RoboDK station: Conveying-with-UR10 (1).rdk

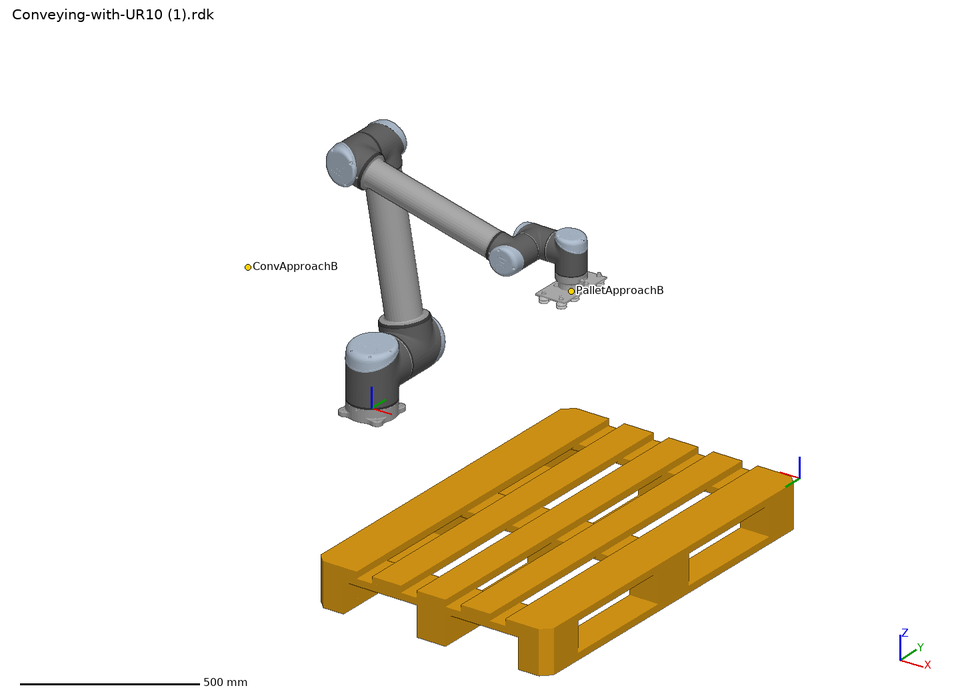
[picture v0: the station drawn from its stored meshes, robots at their saved joint values, targets as dots, program paths as lines]
Station Conveying with UR10 (saved by RoboDK 6.0.5). Poses are relative to the parent item; angles as X-Y-Z fixed-axis rotations.
Station parameters (name, value as stored): SizeBox, 150, 200, 150, SizePallet, 3,2,3, ConvSpeed, 25.0, SENSOR, 0
  - notes Description: <!DOCTYPE HTML PUBLIC "-//W3C//DTD HTML 4.0//EN" "http://www.w3.org/TR/REC-html40/strict.dtd">
<html><head><meta name="qrichtext" content="1" /><style type="text/css">
p, li { white-space: pre-wrap; }
</style></head><body style=" font-family:'MS Shell Dlg 2'; font-size:8.25pt; font-weight:400; font-style:normal;">
<p style=" margin-top:0px; margin-bottom:0px; margin-left:0px; margin-right:0px; -qt-block-indent:0; text-indent:0px;">This example demonstrates a dual-robot pick-and-place application using two collaborative 6-axis UR10 robots equipped with suction cup grippers. The first robot picks cubes from a pallet and places them onto a continuously moving conveyor. The second robot picks the cubes from the conveyor and places them onto another pallet. A Python script developed with the RoboDK API simulates the detection of the cubes on the moving conveyor before the second robot performs the pick operation.</p></body></html>
  - frame UR10 Base B at (1478.64, 1242.75, 0) mm
    - robot UR10 B (model UR10): 6 axes, payload 10 kg, reach 1300 mm, repeatability 0.1 mm, weight 28.9 kg
        modified DH rows (alpha deg, a mm, theta deg, d mm): 0, 0, 0, 118; 90, 0, 180, 0; 0, 612.7, 0, 0; 0, 571.6, 0, 163.9; -90, 0, 0, 115.7; 90, 0, 180, 92.2
        joint limits [-360, -360, -360, -360, -360, -360] to [360, 360, 360, 360, 360, 360]; home [0, -90, 90, -90, -90, 0]; saved at [-180.64, -99.905, 114.086, -104.182, -90, 0]
      - tool GripperB, TCP at (0, 0, 30) mm, rotated rx 0 ry 0 rz 90 deg, size 209.9 x 42 x 100 mm, geometry from test.iges
    - target ConvApproachB (joint target) at (-305.88, -163.9, 417.02) mm, rotated rx -180 ry 0 rz 0 deg; joints [0, -128.114, 134.225, -96.111, -90, 0] of UR10 B
    - target PalletApproachB (joint target) at (566.28, 157.58, 459.33) mm, rotated rx -180 ry 0 rz 179.36 deg; joints [-180.64, -99.905, 114.086, -104.182, -90, 0] of UR10 B
    - frame PalletB at (1034.81, 598.47, -166.38) mm, rotated rx 0 ry 0 rz 179.17 deg
      - object Europallet at (0, 0, 0) mm, size 800 x 144 x 1200 mm, geometry from UUID&
  - program MoveConveyor (1 instructions, listed below)
  - program MainSimulation (5 instructions, listed below)
  - Python program PalletizePreview (listed below)
  - Python program PrepareSimulation (listed below)
  - Python program RobotA_GetParts (listed below)
  - Python program RobotB_StoreParts (listed below)
  - Python program SensorActivate (listed below)
  - Python program SetSimulationParams (listed below)

--- program MoveConveyor ---
  MoveJ (ConveyorMove) [its target is no longer in the station]

--- program MainSimulation ---
  Call PrepareSimulation
  Run MoveConveyor
  Run RobotA_GetParts
  Run SensorActivate
  Call RobotB_StoreParts

--- Python program PalletizePreview ---
# PalletizePreview — roda DENTRO do RoboDK e paletiza com ciclo pick -> place real.
#
# O pick e feito na ESTEIRA (Get Conveyor / ConvApproach), do lado oposto ao pallet, como no
# RobotB_StoreParts.py: a caixa surge sobre a esteira, o robo PEGA (a caixa segue a garra),
# leva ao pallet e SOLTA, camada por camada. Padroes (grid/brick/pinhole/split_block) sao os
# mesmos de palletizer/planner/patterns.py.
#
# COMO RODAR: arraste este arquivo para a janela do RoboDK (ou Tools > Run Script) e Play.

from robodk import robolink, robomath

# ----------------------------- AJUSTE AQUI -----------------------------
PATTERN = "brick"        # "grid" | "brick" | "pinhole" | "split_block"
LAYERS = 4               # no de camadas (minimo 2)
ROBOT_LETTER = "B"       # "A" ou "B" (qual UR10 da estacao)
MOVE_ROBOT = True        # False = so preenche o pallet, sem pick nem robo
APPROACH = 100.0         # folga de aproximacao vertical (mm)

# Nomes da esteira na estacao (fonte do pick). Ajuste se forem diferentes.
CONV_FRAME = "ConveyorReference"
CONV_TARGET = "Get Conveyor"        # ponto de coleta sobre a esteira
CONV_APPROACH = "ConvApproach"      # + letra do robo (ex.: ConvApproachB)

# Fallback (usado SO se a esteira nao for encontrada): pick ao lado do pallet.
PICK_DX = None           # None = centro do pallet em X
PICK_DY = -150.0
# -----------------------------------------------------------------------

RDK = robolink.Robolink()
RDK.setRunMode(robolink.RUNMODE_SIMULATE)


# =========== padroes de amarracao (espelho de planner/patterns.py) ===========
def _base_grid(nx, ny, bx, by):
    return [((i + 0.5) * bx, (j + 0.5) * by, 0.0)
            for j in range(ny) for i in range(nx)]


def layer_positions(pattern, nx, ny, bx, by, layer):
    pos = _base_grid(nx, ny, bx, by)
    if pattern == "brick":
        if layer % 2 == 1:
            pos = [(x + bx / 2.0, y, r) for (x, y, r) in pos]
    elif pattern == "pinhole":
        center = round((ny - 1) / 2.0) * nx + round((nx - 1) / 2.0)
        pos = [p for k, p in enumerate(pos) if k != center]
        if layer % 2 == 1:
            pos = [(x, y, (r + 90.0) % 180.0) for (x, y, r) in pos]
    elif pattern == "split_block":
        mid = nx / 2.0
        pos = [(x, y, 90.0 if ((k % nx < mid) == (layer % 2 == 1)) else 0.0)
               for k, (x, y, r) in enumerate(pos)]
    return pos


# =========== geometria a partir dos params da estacao ===========
def _parse_triplet(value, default):
    try:
        parts = [float(v.replace(" ", "")) for v in str(value).split(",")]
        if len(parts) >= 3:
            return parts[:3]
    except Exception:
        pass
    return default


BX, BY, BZ = _parse_triplet(RDK.getParam("SizeBox"), [100.0, 100.0, 100.0])
size_pallet = _parse_triplet(RDK.getParam("SizePallet"), [3.0, 3.0, float(LAYERS)])
NX, NY = int(size_pallet[0]), int(size_pallet[1])


# =========== itens da estacao ===========
suffix = ROBOT_LETTER.upper()
robot = RDK.Item("UR10 " + suffix, robolink.ITEM_TYPE_ROBOT)
tool = RDK.Item("Gripper" + suffix, robolink.ITEM_TYPE_TOOL)
frame_pallet = RDK.Item("Pallet" + suffix, robolink.ITEM_TYPE_FRAME)
target_safe = RDK.Item("PalletApproach" + suffix, robolink.ITEM_TYPE_TARGET)
partref = RDK.Item("box100mm")

for label, item in [("UR10 " + suffix, robot), ("Pallet" + suffix, frame_pallet),
                    ("box100mm", partref)]:
    if not item.Valid():
        raise Exception("Item '%s' nao encontrado na estacao. Ajuste os nomes no topo." % label)

# esteira (fonte do pick)
frame_conv = RDK.Item(CONV_FRAME, robolink.ITEM_TYPE_FRAME)
target_conv = RDK.Item(CONV_TARGET, robolink.ITEM_TYPE_TARGET)
conv_safe = RDK.Item(CONV_APPROACH + suffix, robolink.ITEM_TYPE_TARGET)
use_conveyor = frame_conv.Valid() and target_conv.Valid()

has_pallet_safe = target_safe.Valid()

# --- define onde e como fazer o pick ---
if use_conveyor:
    pick_frame = frame_conv
    pick_safe = conv_safe if conv_safe.Valid() else None
    pick_tool = target_conv.Pose() * robomath.transl(0, 0, -BZ / 2.0)  # pose de coleta na esteira
    box_local = robomath.transl(*pick_tool.Pos())                      # caixa upright sobre a esteira
    print("Pick: ESTEIRA ('%s')." % CONV_TARGET)
else:
    pick_frame = frame_pallet
    pick_safe = target_safe if has_pallet_safe else None
    px = (NX * BX / 2.0) if PICK_DX is None else PICK_DX
    pick_tool = robomath.transl(px, PICK_DY, BZ / 2.0) * robomath.rotx(robomath.pi)
    box_local = robomath.transl(px, PICK_DY, BZ / 2.0)
    print("Pick: esteira nao encontrada; usando ponto ao lado do pallet (%.0f, %.0f)."
          % (px, PICK_DY))

pick_app = pick_tool * robomath.transl(0, 0, -(APPROACH + BZ))


# =========== limpa caixas anteriores ===========
RDK.Render(False)
for obj in RDK.ItemList(robolink.ITEM_TYPE_OBJECT, False):
    if obj.Name().startswith("Caixa "):
        obj.Delete()
partref.Copy()

if MOVE_ROBOT and tool.Valid():
    robot.setPoseTool(tool)


# =========== helpers ===========
def new_box(index, layer):
    part = frame_pallet.Paste()
    part.Scale([BX / 100.0, BY / 100.0, BZ / 100.0])
    part.setName("Caixa %d" % index)
    part.Recolor([0.2, 0.5, 0.2 + 0.6 * (layer % 2), 1])
    part.setVisible(True, False)
    return part


def rotz(deg):
    return robomath.rotz(robomath.pi * deg / 180.0)


def snap(part, x, y, z, rot_z):
    part.setParentStatic(frame_pallet)
    part.setPose(robomath.transl(x, y, z) * rotz(rot_z))


# =========== execucao ===========
count = 0
reach_fail = 0
first_error_shown = False
for layer in range(LAYERS):
    z_center = (layer + 0.5) * BZ
    for (x, y, rot_z) in layer_positions(PATTERN, NX, NY, BX, BY, layer):
        count += 1
        part = new_box(count, layer)

        if not MOVE_ROBOT:
            snap(part, x, y, z_center, rot_z)
            continue

        # a caixa surge no ponto de coleta (esteira)
        part.setParent(pick_frame)
        part.setPose(box_local)
        RDK.Render(True)

        place = robomath.transl(x, y, z_center) * robomath.rotx(robomath.pi) * rotz(rot_z)
        place_app = place * robomath.transl(0, 0, -(APPROACH + BZ))

        try:
            # PEGA na esteira
            robot.setPoseFrame(pick_frame)
            if pick_safe is not None:
                robot.MoveJ(pick_safe)
            robot.MoveJ(pick_app)
            robot.MoveL(pick_tool)
            part.setParentStatic(tool)      # anexa a caixa a garra
            robot.MoveL(pick_app)
            # SOLTA no pallet
            robot.setPoseFrame(frame_pallet)
            if has_pallet_safe:
                robot.MoveJ(target_safe)
            robot.MoveJ(place_app)
            robot.MoveL(place)
            snap(part, x, y, z_center, rot_z)  # encaixa exato
            robot.MoveL(place_app)
        except Exception as exc:
            reach_fail += 1
            snap(part, x, y, z_center, rot_z)
            if not first_error_shown:
                print("ERRO de movimento na caixa %d: %s" % (count, exc))
                print("  -> verifique alcance do pick/place ou os nomes da esteira no topo.")
                first_error_shown = True

if MOVE_ROBOT and has_pallet_safe:
    try:
        robot.setPoseFrame(frame_pallet)
        robot.MoveJ(target_safe)
    except Exception:
        pass

RDK.Render(True)
print("Padrao '%s': %d caixas, %d camada(s), %d falha(s) de alcance."
      % (PATTERN, count, LAYERS, reach_fail))

--- Python program PrepareSimulation ---
# Type help("robodk.robolink") or help("robodk.robomath") for more information
# Press F5 to run the script
# Documentation: https://robodk.com/doc/en/RoboDK-API.html
# Reference:     https://robodk.com/doc/en/PythonAPI/robodk.html
# Note: It is not required to keep a copy of this file, your Python script is saved with your RDK project

# You can also use the new version of the API:
from robodk import robolink    # RoboDK API
from robodk import robomath    # Robot toolbox
RDK = robolink.Robolink()

# Forward and backwards compatible use of the RoboDK API:
# Remove these 2 lines to follow python programming guidelines
from robodk import *      # RoboDK API
from robolink import *    # Robot toolbox
# Link to RoboDK
# RDK = Robolink()
# Type help("robolink") or help("robodk") for more information
# Press F5 to run the script
# Note: you do not need to keep a copy of this file, your python script is saved with the station

# Use RoboDK API as RL

frame_pallet        = RDK.Item('PalletA', robolink.ITEM_TYPE_FRAME)

# get variable parameters
SIZE_BOX = RDK.getParam('SizeBox')
SIZE_PALLET = RDK.getParam('SizePallet')
SIZE_BOX_XYZ = [float(x.replace(' ','')) for x in SIZE_BOX.split(',')]
SIZE_PALLET_XYZ = [float(x.replace(' ','')) for x in SIZE_PALLET.split(',')]
SIZE_BOX_Z = SIZE_BOX_XYZ[2] # the height of the boxes is important to take into account when approaching the positions

def box_calc(size_xyz, pallet_xyz):
    """Calculates a list of points to store parts in a pallet"""
    [size_x, size_y, size_z] = size_xyz
    [pallet_x, pallet_y, pallet_z] = pallet_xyz
    xyz_list = []
    for h in range(int(pallet_z)):
        for j in range(int(pallet_y)):
            for i in range(int(pallet_x)):
                xyz_list = xyz_list + [[(i+0.5)*size_x, (j+0.5)*size_y, (h+0.5)*size_z]]
    return xyz_list

def parts_setup(frame, positions, size_xyz):
    """Place a list of parts in a reference frame. The part/reference object must have been previously copied to the clipboard."""
    [size_x, size_y, size_z] = size_xyz
    nparts = len(positions)
    cstep = 1.0/(nparts - 1)
    for i in range(nparts):
        newpart = frame.Paste()
        newpart.Scale([size_x/100, size_y/100, size_z/100]) #scale with respect to the reference object (100mm cube)
        newpart.setName('Part ' + str(i+1)) #set item name
        newpart.setPose(robomath.transl(positions[i])) #set item position with respect to parent
        newpart.setVisible(True, False) #make item visible but hide the reference frame
        newpart.Recolor([1-cstep*i, cstep*i, 0.2, 1]) #set RGBA color

def cleanup(objects, startswith="Part "):
    """Deletes all objects where the name starts with "startswith", from the provided list of objects."""
    for item in objects:
        if item.Name().startswith(startswith):
            item.Delete()

# turn off rendering (much faster when setting up the station)
RDK.Render(False)

# cleanup previous simulation (generated parts and tools)
all_objects = RDK.ItemList(robolink.ITEM_TYPE_OBJECT, False)
cleanup(all_objects, 'Part ')
all_tools = RDK.ItemList(robolink.ITEM_TYPE_TOOL, False)
cleanup(all_tools, 'TCP ')

# copy the reference part
partref = RDK.Item('box100mm')
partref.Copy()

#RL.Set_Simulation_Speed(500);
#RL.Set_Simulation_Mode(1)

# calculate an array of positions to get/store the parts
parts_positions = box_calc(SIZE_BOX_XYZ, SIZE_PALLET_XYZ)

# setup/initialise the parts on the palled
parts_setup(frame_pallet, parts_positions, SIZE_BOX_XYZ)

RDK.Render(True)

--- Python program RobotA_GetParts ---
# Type help("robodk.robolink") or help("robodk.robomath") for more information
# Press F5 to run the script
# Documentation: https://robodk.com/doc/en/RoboDK-API.html
# Reference:     https://robodk.com/doc/en/PythonAPI/robodk.html
# Note: It is not required to keep a copy of this file, your Python script is saved with your RDK project

# You can also use the new version of the API:
from robodk import robolink    # RoboDK API
from robodk import robomath    # Robot toolbox
RDK = robolink.Robolink()

# Forward and backwards compatible use of the RoboDK API:
# Remove these 2 lines to follow python programming guidelines
from robodk import *      # RoboDK API
from robolink import *    # Robot toolbox
# Link to RoboDK
# RDK = Robolink()
# Type help("robolink") or help("robodk") for more information
# Press F5 to run the script
# Note: you do not need to keep a copy of this file, your python script is saved with the station

# Use RoboDK API as RL

# define default approach distance
APPROACH = 100

# gather robot, tool and reference frames from the station
robot               = RDK.Item('UR10 A', robolink.ITEM_TYPE_ROBOT)
tool                = RDK.Item('GripperA', robolink.ITEM_TYPE_TOOL)
frame_pallet        = RDK.Item('PalletA', robolink.ITEM_TYPE_FRAME)
frame_conv          = RDK.Item('ConveyorReference', robolink.ITEM_TYPE_FRAME)
frame_conv_moving   = RDK.Item('MovingRef', robolink.ITEM_TYPE_FRAME)

# gather targets
target_pallet_safe = RDK.Item('PalletApproachA', robolink.ITEM_TYPE_TARGET)
target_conv_safe = RDK.Item('ConvApproachA', robolink.ITEM_TYPE_TARGET)
target_conv = RDK.Item('Put Conveyor', robolink.ITEM_TYPE_TARGET)

# get variable parameters
SIZE_BOX = RDK.getParam('SizeBox')
SIZE_PALLET = RDK.getParam('SizePallet')
SIZE_BOX_XYZ = [float(x.replace(' ','')) for x in SIZE_BOX.split(',')]
SIZE_PALLET_XYZ = [float(x.replace(' ','')) for x in SIZE_PALLET.split(',')]
SIZE_BOX_Z = SIZE_BOX_XYZ[2] # the height of the boxes is important to take into account when approaching the positions

def box_calc(size_xyz, pallet_xyz):
    """Calculates a list of points to store parts in a pallet"""
    [size_x, size_y, size_z] = size_xyz
    [pallet_x, pallet_y, pallet_z] = pallet_xyz
    xyz_list = []
    for h in range(int(pallet_z)):
        for j in range(int(pallet_y)):
            for i in range(int(pallet_x)):
                xyz_list = xyz_list + [[(i+0.5)*size_x, (j+0.5)*size_y, (h+0.5)*size_z]]
    return xyz_list

def TCP_On(toolitem):
    """Attaches the closest object to the toolitem Htool pose,
    It will also output appropriate function calls on the generated robot program (call to TCP_On)"""
    toolitem.AttachClosest()
    toolitem.RDK().RunMessage('Set air valve on')
    toolitem.RDK().RunProgram('TCP_On()');

def TCP_Off(toolitem, itemleave=0):
    """Detaches the closest object attached to the toolitem Htool pose,
    It will also output appropriate function calls on the generated robot program (call to TCP_Off)"""
    toolitem.DetachAll(itemleave)
    toolitem.RDK().RunMessage('Set air valve off')
    toolitem.RDK().RunProgram('TCP_Off()');

#RL.Set_Simulation_Speed(500);
#RL.Set_Simulation_Mode(1)

# calculate an array of positions to get/store the parts
parts_positions = box_calc(SIZE_BOX_XYZ, SIZE_PALLET_XYZ)

# Calculate a new TCP that takes into account the size of the part (targets are set to the center of the box)
tool_xyzrpw = tool.PoseTool()*robomath.transl(0,0,SIZE_BOX_Z/2)
tool_tcp = robot.AddTool(tool_xyzrpw, 'TCP A')

# ---------------------------------------------------------------------------------
# -------------------------- PROGRAM START ----------------------------------------

robot.setPoseTool(tool_tcp)
nparts = len(parts_positions)
i = nparts-1
while i >= 0:
    # ----------- take a part from the pallet ------
    # get the xyz position of part i
    robot.setPoseFrame(frame_pallet)
    part_position_i = parts_positions[i]
    target_i = robomath.transl(part_position_i)*robomath.rotx(pi)
    target_i_app = target_i * robomath.transl(0,0,-(APPROACH+SIZE_BOX_Z))
    # approach to the pallet
    robot.MoveJ(target_pallet_safe)
    # get the box i
    robot.MoveJ(target_i_app)
    robot.MoveL(target_i)
    TCP_On(tool) # attach the closest part
    robot.MoveL(target_i_app)
    robot.MoveJ(target_pallet_safe)

    # ----------- place the box i on the convegor ------
    # approach to the conveyor
    robot.setPoseFrame(frame_conv)
    target_conv_pose = target_conv.Pose()*robomath.transl(0,0,-SIZE_BOX_Z/2)
    target_conv_app = target_conv_pose*robomath.transl(0,0,-APPROACH)
    robot.MoveJ(target_conv_safe)
    robot.MoveJ(target_conv_app)
    robot.MoveL(target_conv_pose)
    TCP_Off(tool, frame_conv_moving) # detach an place the object in the moving reference frame of the conveyor
    robot.MoveL(target_conv_app)
    robot.MoveJ(target_conv_safe)

    i = i - 1

--- Python program RobotB_StoreParts ---
# Type help("robodk.robolink") or help("robodk.robomath") for more information
# Press F5 to run the script
# Documentation: https://robodk.com/doc/en/RoboDK-API.html
# Reference:     https://robodk.com/doc/en/PythonAPI/robodk.html
# Note: It is not required to keep a copy of this file, your Python script is saved with your RDK project

# You can also use the new version of the API:
from robodk import robolink    # RoboDK API
from robodk import robomath    # Robot toolbox
RDK = robolink.Robolink()

# Forward and backwards compatible use of the RoboDK API:
# Remove these 2 lines to follow python programming guidelines
from robodk import *      # RoboDK API
from robolink import *    # Robot toolbox
# Link to RoboDK
# RDK = Robolink()
# Type help("robolink") or help("robodk") for more information
# Press F5 to run the script
# Note: you do not need to keep a copy of this file, your python script is saved with the station

# Use RoboDK API as RL

# define default approach distance
APPROACH = 100
SENSOR_VARIABLE = 'SENSOR' # station variable

# gather robot, tool and reference frames from the station
robot               = RDK.Item('UR10 B', robolink.ITEM_TYPE_ROBOT)
tool                = RDK.Item('GripperB', robolink.ITEM_TYPE_TOOL)
frame_pallet        = RDK.Item('PalletB', robolink.ITEM_TYPE_FRAME)
frame_conv          = RDK.Item('ConveyorReference', robolink.ITEM_TYPE_FRAME)
frame_conv_moving   = RDK.Item('MovingRef', robolink.ITEM_TYPE_FRAME)

# gather targets
target_pallet_safe = RDK.Item('PalletApproachB', robolink.ITEM_TYPE_TARGET)
target_conv_safe = RDK.Item('ConvApproachB', robolink.ITEM_TYPE_TARGET)
target_conv = RDK.Item('Get Conveyor', robolink.ITEM_TYPE_TARGET)

# get variable parameters
SIZE_BOX = RDK.getParam('SizeBox')
SIZE_PALLET = RDK.getParam('SizePallet')
SIZE_BOX_XYZ = [float(x.replace(' ','')) for x in SIZE_BOX.split(',')]
SIZE_PALLET_XYZ = [float(x.replace(' ','')) for x in SIZE_PALLET.split(',')]
SIZE_BOX_Z = SIZE_BOX_XYZ[2] # the height of the boxes is important to take into account when approaching the positions

def box_calc(size_xyz, pallet_xyz):
    """Calculates a list of points to store parts in a pallet"""
    [size_x, size_y, size_z] = size_xyz
    [pallet_x, pallet_y, pallet_z] = pallet_xyz
    xyz_list = []
    for h in range(int(pallet_z)):
        for j in range(int(pallet_y)):
            for i in range(int(pallet_x)):
                xyz_list = xyz_list + [[(i+0.5)*size_x, (j+0.5)*size_y, (h+0.5)*size_z]]
    return xyz_list

def TCP_On(toolitem):
    """Attaches the closest object to the toolitem Htool pose,
    It will also output appropriate function calls on the generated robot program (call to TCP_On)"""
    toolitem.AttachClosest()
    toolitem.RDK().RunMessage('Set air valve on')
    toolitem.RDK().RunProgram('TCP_On()');

def TCP_Off(toolitem, itemleave=0):
    """Detaches the closest object attached to the toolitem Htool pose,
    It will also output appropriate function calls on the generated robot program (call to TCP_Off)"""
    #toolitem.DetachClosest(itemleave)
    toolitem.DetachAll(itemleave)
    toolitem.RDK().RunMessage('Set air valve off')
    toolitem.RDK().RunProgram('TCP_Off()');

# calculate an array of positions to get/store the parts
parts_positions = box_calc(SIZE_BOX_XYZ, SIZE_PALLET_XYZ)

# Calculate a new TCP that takes into account the size of the part (targets are set to the center of the box)
tool_xyzrpw = tool.PoseTool()*robomath.transl(0,0,SIZE_BOX_Z/2)
tool_tcp = robot.AddTool(tool_xyzrpw, 'TCP B')

# ---------------------------------------------------------------------------------
# -------------------------- PROGRAM START ----------------------------------------

def WaitSensor():
    if RDK.RunMode() == robolink.RUNMODE_SIMULATE:
        # Simulate the sensor by waiting for the SENSOR status to turn to 1 (object present)
        while RDK.getParam(SENSOR_VARIABLE) == 0:
            pause(0.001)
    else:
        RDK.RunProgram('WaitSensor')
    print("Part detected")

robot.setPoseTool(tool_tcp)
nparts = len(parts_positions)
i = 0
while i < nparts:
    # ----------- place the box i on the convegor ------
    # approach to the conveyor
    robot.setPoseFrame(frame_conv)
    target_conv_pose = target_conv.Pose()*robomath.transl(0,0,-SIZE_BOX_Z/2)
    target_conv_app = target_conv_pose*robomath.transl(0,0,-APPROACH)
    robot.MoveJ(target_conv_safe)
    robot.MoveJ(target_conv_app)
    WaitSensor()
    robot.MoveL(target_conv_pose)
    TCP_On(tool) # detach an place the object in the moving reference frame of the conveyor
    robot.MoveL(target_conv_app)
    robot.MoveJ(target_conv_safe)

    # ----------- take a part from the conveyor ------
    # get the xyz position of part i
    robot.setPoseFrame(frame_pallet)
    part_position_i = parts_positions[i]
    target_i = robomath.transl(part_position_i)*robomath.rotx(pi)
    target_i_app = target_i * robomath.transl(0,0,-(APPROACH+SIZE_BOX_Z))
    # approach to the pallet
    robot.MoveJ(target_pallet_safe)
    # get the box i
    robot.MoveJ(target_i_app)
    robot.MoveL(target_i)
    TCP_Off(tool, frame_pallet) # attach the closest part
    robot.MoveL(target_i_app)
    robot.MoveJ(target_pallet_safe)

    i = i + 1

--- Python program SensorActivate ---
# Type help("robodk.robolink") or help("robodk.robomath") for more information
# Press F5 to run the script
# Documentation: https://robodk.com/doc/en/RoboDK-API.html
# Reference:     https://robodk.com/doc/en/PythonAPI/robodk.html
# Note: It is not required to keep a copy of this file, your Python script is saved with your RDK project

# You can also use the new version of the API:
from robodk import robolink    # RoboDK API
from robodk import robomath    # Robot toolbox
RDK = robolink.Robolink()

# Forward and backwards compatible use of the RoboDK API:
# Remove these 2 lines to follow python programming guidelines
from robodk import *      # RoboDK API
from robolink import *    # Robot toolbox
# Link to RoboDK
# RDK = Robolink()
# Type help("robolink") or help("robodk") for more information
# Press F5 to run the script
# Note: you do not need to keep a copy of this file, your python script is saved with the station

# This script allows to simulate a laser sensor
# that detect the presence of a part in a plane,
# such as a part crossing a laser sensor in a
# conveyor belt

# Use a target from the station as a reference plane:
SENSOR_NAME = 'Sensor SICK WL4S'
SENSOR_VARIABLE = 'SENSOR'

# Look for parts with the keyword "Part"
PART_KEYWORD = 'Part '

# Update status every 1 ms
RECHECK_PERIOD = 0.001

# Get the sensor and the detection plane
SENSOR = RDK.Item(SENSOR_NAME, robolink.ITEM_TYPE_OBJECT)

# retrieve all objects
all_objects = RDK.ItemList(robolink.ITEM_TYPE_OBJECT, False)
part_objects = []
for obj in all_objects:
    if obj.Name().count(PART_KEYWORD) > 0:
        part_objects.append(obj)


# Loop forever to detect parts
detected_status = -1
while True:
    detected = 0
    for obj in part_objects:
        # check if an object has the part keyword and is detected by the laser
        if SENSOR.Collision(obj) > 0:
            detected = 1
            break

    # update the current status of the sensor
    if detected_status != detected:
        detected_status = detected
        RDK.setParam(SENSOR_VARIABLE, detected_status)
        print('Object detected status --> %i' % detected_status)

    # Wait some time...
    pause(RECHECK_PERIOD)

--- Python program SetSimulationParams ---
# Type help("robodk.robolink") or help("robodk.robomath") for more information
# Press F5 to run the script
# Documentation: https://robodk.com/doc/en/RoboDK-API.html
# Reference:     https://robodk.com/doc/en/PythonAPI/robodk.html
# Note: It is not required to keep a copy of this file, your Python script is saved with your RDK project

# You can also use the new version of the API:
from robodk import robolink    # RoboDK API
from robodk import robomath    # Robot toolbox
RDK = robolink.Robolink()

# Forward and backwards compatible use of the RoboDK API:
# Remove these 2 lines to follow python programming guidelines
from robodk import *      # RoboDK API
from robolink import *    # Robot toolbox
# Link to RoboDK
# RDK = Robolink()
# Type help("robolink") or help("robodk") for more information
# Press F5 to run the script
# Note: you do not need to keep a copy of this file, your python script is saved with the station


PARAM_SIZE_BOX = 'SizeBox'
PARAM_SIZE_PALLET = 'SizePallet'
PARAM_CONV_SPEED_MM = 'ConvSpeed'




size_box = RDK.getParam(PARAM_SIZE_BOX)
size_pallet = RDK.getParam(PARAM_SIZE_PALLET)
conv_speed = RDK.getParam(PARAM_CONV_SPEED_MM)

# ------------------------------------------------------------
size_box_input = mbox('Enter the size of the box in mm [L,W,H]', entry=size_box)
if size_box_input:
    RDK.setParam(PARAM_SIZE_BOX, size_box_input)
else:
    raise Exception('Operation cancelled by user')

# ------------------------------------------------------------
size_pallet_input = mbox('Enter the size of the pallet', entry=size_pallet)
if size_pallet_input:
    RDK.setParam(PARAM_SIZE_PALLET, size_pallet_input)
else:
    raise Exception('Operation cancelled by user')

# ------------------------------------------------------------
conv_speed_input = mbox('Enter the speed of the conveyor in mm/s', entry=conv_speed)
if conv_speed_input:
    RDK.setParam(PARAM_CONV_SPEED_MM, conv_speed_input)
    conv_speed = float(conv_speed_input)
    conv = RDK.Item('Conveyor Belt', robolink.ITEM_TYPE_ROBOT)
    conv.setSpeed(conv_speed)

else:
    raise Exception('Operation cancelled by user')
